TYPE "MEStoPLC_Common"
VERSION : 0.1
   STRUCT
      "M-MesOnline" : Bool;
      "M-HeartBeat" : Bool;
      Reserve : Array[1..197] of Byte;
   END_STRUCT;

END_TYPE

